// Mitsubishi GX Works2 project: monitort   PLC: Q03UDV

PROGRAM MAIN
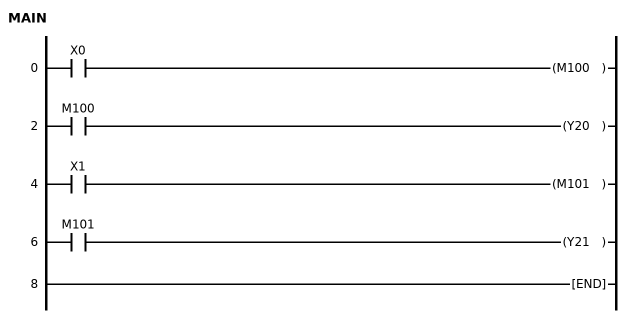
0     LD      X0
      OUT     M100
2     LD      M100
      OUT     Y20
4     LD      X1
      OUT     M101
6     LD      M101
      OUT     Y21
8     END
END_PROGRAM
